RoboDK station: New Station (2).rdk

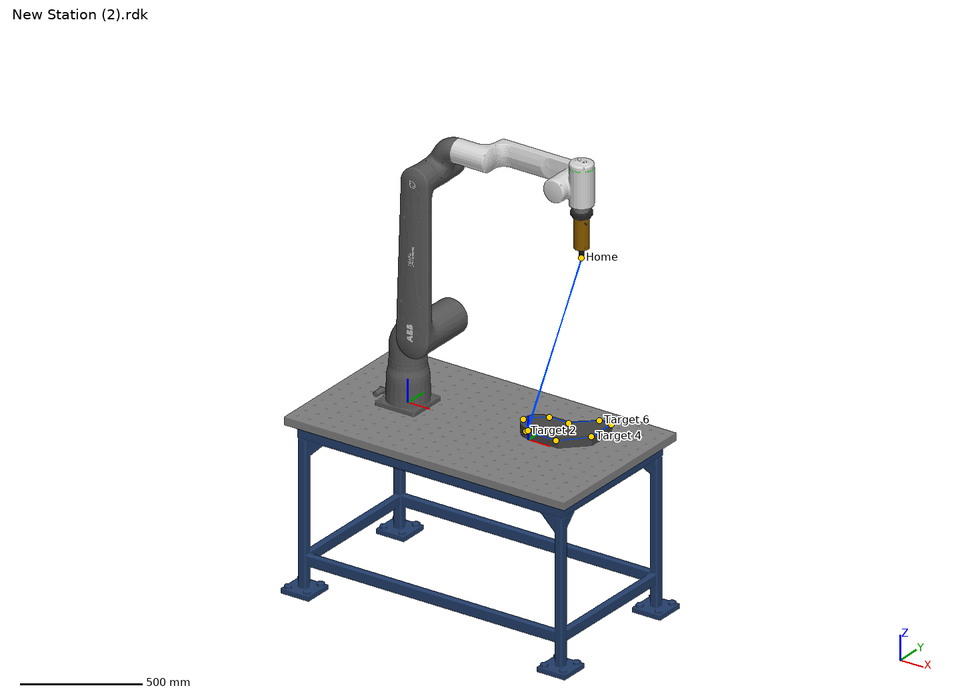
[picture v0: the station drawn from its stored meshes, robots at their saved joint values, targets as dots, program paths as lines]
Station New Station (2) (saved by RoboDK 5.9.2). Poses are relative to the parent item; angles as X-Y-Z fixed-axis rotations.
  - frame ABB CRB 15000 10 Base at (0, 0, 0) mm
    - robot ABB CRB 15000 10: 6 axes
        modified DH rows (alpha deg, a mm, theta deg, d mm): 0, 0, 0, 400; -90, 150, -90, 0; 0, 707, 0, 0; -90, 110, 0, 637; 90, 0, 0, 0; -90, 80, 180, 101
        joint limits [-270, -180, -225, -180, -180, -270] to [270, 180, 85, 180, 180, 270]; home [0, 0, 0, 0, 0, 0]; saved at [0, 0, 0, 0, 90, 0]
      - tool ATI 9150-CDB-8-11-000 Deburring Tool (Spring), TCP at (0, 0, 215) mm, size 93.7 x 93.7 x 214.4 mm
    - object Table 1400x800x800mm at (0, 0, 0) mm, size 1420 x 820 x 800 mm, geometry from Table-1400x800x800mm.sld
  - frame Frame 2 at (600, 0, 0) mm
    - object random1 at (0, 0, 0) mm, size 325 x 240 x 50 mm, geometry from random1.step
    - target Home (Cartesian target) at (267, 0, 901) mm, rotated rx 180 ry 0 rz -180 deg; joints [0, 0, 0, 0, 90, 0] of ABB CRB 15000 10
    - target Target 2 (Cartesian target) at (-3, -10, 41) mm, rotated rx 180 ry 0 rz 180 deg; joints [-0.96, 31.405, 68.51, 0, -9.915, -0.96] of ABB CRB 15000 10
    - target Target 3 (Cartesian target) at (147, -10, 41) mm, rotated rx 180 ry 0 rz 180 deg; joints [-0.767, 33.353, 54.991, 0, 1.656, -0.767] of ABB CRB 15000 10
    - target Target 4 (Cartesian target) at (247, 100, 41) mm, rotated rx 180 ry 0 rz -180 deg; joints [6.733, 36.254, 45.074, 0, 8.672, 6.733] of ABB CRB 15000 10
    - target Target 5 (Cartesian target) at (247, 240, 41) mm, rotated rx 180 ry 0 rz 180 deg; joints [15.82, 37.142, 42.431, 0, 10.426, 15.82] of ABB CRB 15000 10
    - target Target 6 (Cartesian target) at (187, 240, 41) mm, rotated rx 180 ry 0 rz -180 deg; joints [16.959, 35.339, 47.936, 0, 6.726, 16.959] of ABB CRB 15000 10
    - target Target 7 (Cartesian target) at (97, 150, 41) mm, rotated rx 180 ry 0 rz 180 deg; joints [12.145, 32.635, 58.112, 0, -0.747, 12.145] of ABB CRB 15000 10
    - target Target 8 (Cartesian target) at (0, 150, 41) mm, rotated rx -180 ry 0 rz -180 deg; joints [14.036, 31.451, 66.611, 0, -8.062, 14.036] of ABB CRB 15000 10
    - target Target 9 (Cartesian target) at (-75, 75, 41) mm, rotated rx 180 ry 0 rz -180 deg; joints [8.13, 32.081, 74.394, 0, -16.475, 8.13] of ABB CRB 15000 10
    - target Target 10 (Cartesian target) at (0, 0, 41) mm, rotated rx 180 ry 0 rz -180 deg; joints [0, 31.405, 68.251, 0, -9.657, 0] of ABB CRB 15000 10
    - target Target 11 (Cartesian target) at (267, 0, 901) mm, rotated rx 180 ry 0 rz -180 deg; joints [0, 0, 0, 0, 90, 0] of ABB CRB 15000 10
  - program Prog2 (13 instructions, listed below)
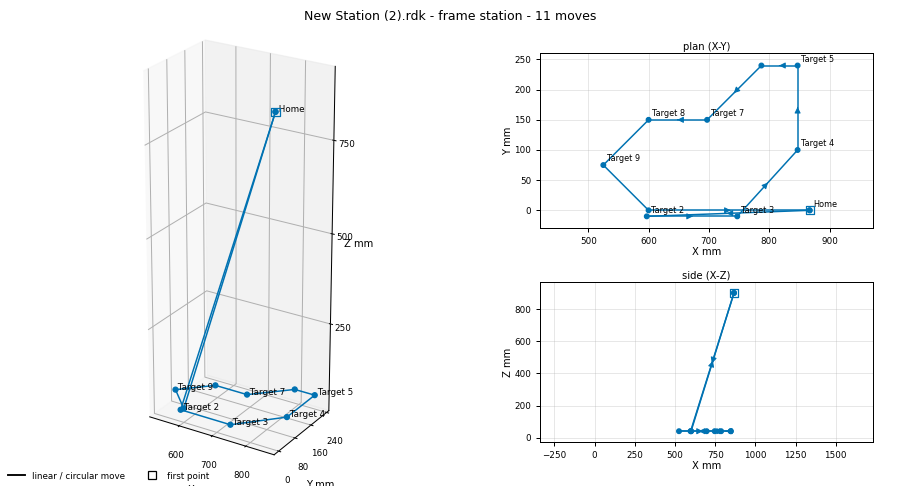
[picture p0: tool path of New Station (2).rdk in frame station, 11 of 11 moves have a stored position in this frame; points joined in program order, loops and branches not executed]

--- program Prog2 (robot ABB CRB 15000 10) ---
  Set Ref.: Frame 2
  Set Tool: ATI 9150-CDB-8-11-000 Deburring Tool (Spring)
  MoveJ (Home)
  MoveL (Target 2)
  MoveL (Target 3)
  MoveL (Target 4)
  MoveL (Target 5)
  MoveL (Target 6)
  MoveL (Target 7)
  MoveL (Target 8)
  MoveC (Target 8, Target 9)
  MoveC (Target 9, Target 10)
  MoveL (Target 11)
